TYPE typeStationLocks :
STRUCT
	Station1Locked:BOOL;
	Station2Locked:BOOL;
	Station3Locked:BOOL;
	Station4Locked:BOOL;
	Station5Locked:BOOL;
	Station6Locked:BOOL;
						
END_STRUCT
END_TYPE

(* stored: Version 1.1.0.1, ProductVersion 3.1.4024.11
   DUT typeStationLocks: Id {696fd29a-3340-03da-31af-06dc555bda12} *)
